(* IEC 61131-3 sources: git_feedingMachine/app/src/_internal, 3 files *)

(* ---- AxisCtrlTypes.st ---- *)
NAMESPACE Siemens.Simatic.Motion

    TYPE
        AxisData : STRUCT
            cmd : AxisCmd;
            enabled : BOOL;
            homed : BOOL;
            error : BOOL;
            errorID : WORD;
            actSpeed : LREAL;
            actVelocity : LREAL;
            actPosition : LREAL;
        END_STRUCT;
    END_TYPE

    TYPE
        AxisCmd : INT (
            NONE := 0,
            ENABLE := 1,
            DISABLE := 2,
            RESET := 3,
            HOME := 4,
            STOP := 5,
            JOG := 6,
            POS_RELATIVE := 7,
            POS_ABSOLUTE := 8) := NONE;
    END_TYPE

END_NAMESPACE

(* ---- PosAxis.st ---- *)
USING Siemens.Simatic.S71500.MotionControl.Native;
NAMESPACE Siemens.Simatic.Motion

    CLASS PUBLIC PosAxis EXTENDS SpeedAxis

        VAR PROTECTED
            _axisAsPos : REF_TO TO_PositioningAxis;
            _mcHome : MC_HOME;
            _mcMoveRel : MC_MOVERELATIVE;
            _mcMoveAbs : MC_MOVEABSOLUTE;
        END_VAR

        METHOD PUBLIC OVERRIDE Attach : BOOL
            VAR_INPUT
                axisDB : DB_ANY;
            END_VAR
            _axisDB := axisDB;
            Attach := THIS.RefToAxisIsValid();
            SUPER.CallMcBlocksSpeedAxis();
            THIS.CallMcBlocksPosAxis();
        END_METHOD

        METHOD PUBLIC OVERRIDE ResetCmds
            SUPER.ResetCmds();
            _mcHome.Execute := FALSE;
            _mcMoveRel.Execute := FALSE;
            _mcMoveAbs.Execute := FALSE;
        END_METHOD

        METHOD PUBLIC HomeAxis
            VAR_INPUT
                position : LREAL;
                homingMode : INT;
            END_VAR
            _mcHome.Mode := homingMode;
            _mcHome.Position := position;
            _mcHome.Execute := TRUE;
            _axisData.cmd := AxisCmd#HOME;
        END_METHOD

        METHOD PUBLIC PosRelative
            VAR_INPUT
                distance : LREAL;
                velocity : LREAL;
                acceleration : LREAL;
                deceleration : LREAL;
                jerk : LREAL;
            END_VAR
            _mcMoveRel.Execute := TRUE;
            _mcMoveRel.Distance := distance;
            _mcMoveRel.velocity := velocity;
            _mcMoveRel.Acceleration := acceleration;
            _mcMoveRel.Deceleration := deceleration;
            _axisData.cmd := AxisCmd#POS_RELATIVE;
        END_METHOD

        METHOD PUBLIC PosAbsolute
            VAR_INPUT
                position : LREAL;
                velocity : LREAL;
                acceleration : LREAL;
                deceleration : LREAL;
                jerk : LREAL;
                direction : INT;
            END_VAR
            _mcMoveAbs.Execute := TRUE;
            _mcMoveAbs.Position := position;
            _mcMoveAbs.velocity := velocity;
            _mcMoveAbs.Acceleration := acceleration;
            _mcMoveAbs.Deceleration := deceleration;
            _mcMoveAbs.Jerk := -1;
            IF direction > 0 THEN
                _mcMoveAbs.Direction := direction;
            ELSE
                _mcMoveAbs.Direction := 1;
            END_IF;
            _axisData.cmd := AxisCmd#POS_ABSOLUTE;
        END_METHOD

        METHOD PUBLIC OVERRIDE GetAxisStatus : AxisData
            _axisData.enabled := _mcPower.Status;
            _axisData.homed := _axisAsPos^.StatusWord.%X5;
            IF _mcPower.Error THEN
                _axisData.error := TRUE;
                _axisData.errorID := _mcPower.ErrorId;
            ELSIF _mcReset.Error THEN
                _axisData.error := TRUE;
                _axisData.errorID := _mcReset.ErrorId;
            ELSIF _mcHalt.Error THEN
                _axisData.error := TRUE;
                _axisData.errorID := _mcHalt.ErrorId;
            ELSIF _mcMoveVel.Error THEN
                _axisData.error := TRUE;
                _axisData.errorID := _mcMoveVel.ErrorId;
            ELSIF _mcHome.Error THEN
                _axisData.error := TRUE;
                _axisData.errorID := _mcHome.ErrorId;
            ELSIF _mcMoveRel.Error THEN
                _axisData.error := TRUE;
                _axisData.errorID := _mcMoveRel.ErrorId;
            ELSIF _mcMoveAbs.Error THEN
                _axisData.error := TRUE;
                _axisData.errorID := _mcMoveAbs.ErrorId;
            ELSE
                _axisData.error := FALSE;
                _axisData.errorID := WORD#16#0000;
            END_IF;
            _axisData.actVelocity := _axisAsPos^.ActualVelocity;
            _axisData.actPosition := _axisAsPos^.ActualPosition;
            GetAxisStatus := _axisData;
        END_METHOD

        METHOD PROTECTED CallMcBlocksPosAxis
            _axisAsPos := AsPositioningAxisRef(_axisDB);
            _axisAsAxis := _axisAsPos;
            IF _axisAsPos <> NULL THEN
                _mcHome(Axis := _axisAsAxis^);
                _mcMoveRel(Axis := _axisAsPos^);
                _mcMoveAbs(Axis := _axisAsPos^);
                IF _mcHome.Done THEN
                    _axisData.cmd := AxisCmd#NONE;
                    _mcHome.Execute := FALSE;
                END_IF;

                IF _mcMoveRel.Done OR _mcMoveRel.CommandAborted THEN
                    _mcMoveRel.Execute := FALSE;
                END_IF;

                IF _mcMoveAbs.Done OR _mcMoveAbs.CommandAborted THEN
                    _mcMoveAbs.Execute := FALSE;
                END_IF;
            ELSE
                RETURN;
            END_IF;
        END_METHOD

        METHOD PROTECTED OVERRIDE RefToAxisIsValid : BOOL
            _axisAsPos := AsPositioningAxisRef(_axisDB);
            RefToAxisIsValid := _axisAsPos <> NULL;
        END_METHOD

    END_CLASS

END_NAMESPACE

(* ---- SpeedAxis.st ---- *)
USING Siemens.Simatic.S71500.MotionControl.Native;
NAMESPACE Siemens.Simatic.Motion

    CLASS PUBLIC SpeedAxis

        VAR PROTECTED
            _axisAsSpeed : REF_TO TO_SpeedAxis;
            _axisAsAxis : REF_TO TO_Axis;
            _mcPower : MC_POWER;
            _mcReset : MC_RESET;
            _mcJog : MC_MOVEJOG;
            _mcHalt : MC_HALT;
            _mcMoveVel : MC_MOVEVELOCITY;
            _axisData : AxisData;
            _axisDB : DB_ANY;
        END_VAR

        METHOD PUBLIC Attach : BOOL
            VAR_INPUT
                axisDB : DB_ANY;
            END_VAR
            _axisDB := axisDB;
            Attach := THIS.RefToAxisIsValid();
            THIS.CallMcBlocksSpeedAxis();
        END_METHOD

        METHOD PUBLIC ResetCmds
            _mcReset.Execute := FALSE;
            _mcHalt.Execute := FALSE;
            _mcMoveVel.Execute := FALSE;
        END_METHOD

        METHOD PUBLIC EnableAxis
            VAR_INPUT
                startMode : INT;
            END_VAR
            _mcPower.StartMode := startMode;
            _mcPower.Enable := TRUE;
            _axisData.cmd := AxisCmd#ENABLE;
        END_METHOD

        METHOD PUBLIC DisableAxis
            VAR_INPUT
                stopMode : INT;
            END_VAR
            _mcPower.StopMode := stopMode;
            _mcPower.Enable := FALSE;
            _axisData.cmd := AxisCmd#DISABLE;
        END_METHOD

        METHOD PUBLIC ResetAxis
                _mcReset.Execute := TRUE;
                _axisData.cmd := AxisCmd#RESET;
                IF _mcReset.Done THEN
                    _axisData.cmd := AxisCmd#NONE;
                    _mcHalt.Execute := FALSE;
                END_IF;
        END_METHOD

        METHOD PUBLIC StopAxis
            VAR_INPUT
                deceleration : LREAL;
                jerk : LREAL;
                abortAcceleration : BOOL;
            END_VAR
            _mcHalt.Deceleration := deceleration;
            _mcHalt.Jerk := jerk;
            _mcHalt.AbortAcceleration := abortAcceleration;
            _mcHalt.Execute := TRUE;
            _axisData.cmd := AxisCmd#STOP;
            IF _mcHalt.Done THEN
                _axisData.cmd := AxisCmd#NONE;
                _mcHalt.Execute := FALSE;
            END_IF;
        END_METHOD

        METHOD PUBLIC MoveVelocity
            VAR_INPUT
                velocity : LREAL;
                acceleration : LREAL;
                deceleration : LREAL;
                jerk : LREAL;
                direction : INT;
                maintainCurrentVel : BOOL;
            END_VAR
            _mcMoveVel.velocity := velocity;
            _mcMoveVel.Acceleration := acceleration;
            _mcMoveVel.Deceleration := deceleration;
            _mcMoveVel.Jerk := jerk;
            _mcMoveVel.direction := direction;
            _mcMoveVel.Current := maintainCurrentVel;
            _mcMoveVel.Execute := TRUE;
            IF _mcMoveVel.CommandAborted THEN
                _axisData.cmd := AxisCmd#NONE;
                _mcMoveVel.Execute := FALSE;
            END_IF;
        END_METHOD

        METHOD PUBLIC GetAxisStatus : AxisData
            _axisData.enabled := _mcPower.Status;
            IF _mcPower.Error THEN
                _axisData.error := TRUE;
                _axisData.errorID := _mcPower.ErrorId;
            ELSIF _mcReset.Error THEN
                _axisData.error := TRUE;
                _axisData.errorID := _mcReset.ErrorId;
            ELSIF _mcHalt.Error THEN
                _axisData.error := TRUE;
                _axisData.errorID := _mcHalt.ErrorId;
            ELSIF _mcMoveVel.Error THEN
                _axisData.error := TRUE;
                _axisData.errorID := _mcMoveVel.ErrorId;
            ELSE
                _axisData.error := FALSE;
                _axisData.errorID := WORD#16#0000;
            END_IF;
            _axisData.actSpeed := _axisAsSpeed^.ActualSpeed;
            GetAxisStatus := _axisData;
        END_METHOD

        METHOD PROTECTED CallMcBlocksSpeedAxis
            IF NOT THIS.RefToAxisIsValid() THEN
                RETURN;
            ELSE
                _axisAsSpeed := AsSpeedAxisRef(_axisDB);
                _axisAsAxis := AsAxisRef(_axisDB);
                _mcPower(Axis := _axisAsAxis^);
                _mcReset(Axis := _axisAsAxis^);
                _mcHalt(Axis := _axisAsSpeed^);
                _mcJog(Axis := _axisAsSpeed^);
                _mcMoveVel(Axis := _axisAsSpeed^);
            END_IF;
        END_METHOD

        METHOD PROTECTED RefToAxisIsValid : BOOL
                _axisAsSpeed := AsSpeedAxisRef(_axisDB);
                RefToAxisIsValid := _axisAsSpeed <> NULL;
        END_METHOD

    END_CLASS

END_NAMESPACE
